FUNCTION_BLOCK POSTGRE_DB_INSERT_JSON_TIMESERIES
  {SET_ATTRIBUTE(OpcUa, POINT.ENDPOINT)}
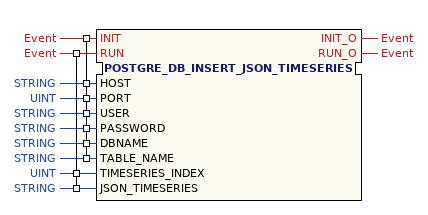
  EVENT_INPUT
    INIT WITH HOST, PORT, USER, PASSWORD, DBNAME, TABLE_NAME;
    RUN WITH TIMESERIES_INDEX, JSON_TIMESERIES;
  END_EVENT
  EVENT_OUTPUT
    INIT_O;
    RUN_O;
  END_EVENT
  VAR_INPUT
    HOST : STRING; {SET_ATTRIBUTE(OpcUa, Constant)}
    PORT : UINT; {SET_ATTRIBUTE(OpcUa, Constant)}
    USER : STRING; {SET_ATTRIBUTE(OpcUa, Constant)}
    PASSWORD : STRING; {SET_ATTRIBUTE(OpcUa, Constant)}
    DBNAME : STRING; {SET_ATTRIBUTE(OpcUa, Constant)}
    TABLE_NAME : STRING; {SET_ATTRIBUTE(OpcUa, Constant)}
    TIMESERIES_INDEX : UINT; {SET_ATTRIBUTE(OpcUa, Constant)}
    JSON_TIMESERIES : STRING; {SET_ATTRIBUTE(OpcUa, Variable.RUN)}
  END_VAR
END_FUNCTION_BLOCK
